FUNCTION_BLOCK fbLichtSensor IMPLEMENTS ITFGesimuleerdDO
VAR_INPUT
END_VAR
VAR_OUTPUT
END_VAR
VAR
	BHmiPalletSensorSim : BOOL;
	sensorwaarde1 : BOOL;
END_VAR

{warning 'Add property implementation'}
PROPERTY SensorWaarde : BOOL
GET
BHmiPalletSensorSim:= SensorWaarde1;
END_GET
SET
SensorWaarde1 := BHmiPalletSensorSim;
END_SET
END_PROPERTY

END_FUNCTION_BLOCK

(* stored: Version 1.1.0.1
   POU fbLichtSensor: Id {2a2763db-7b58-400d-b689-256626899efb}, SpecialFunc None
   Property SensorWaarde: Id {ceea8ccb-d715-4f5f-bef2-cc7a9aa76013}
   Get Get: Id {2a076388-55d1-4080-9c55-60bdd5547358}
   Set Set: Id {b3401fe1-3921-4ebe-bc43-cea8512b372a} *)
